///////////
// Structure for CtrlPcs Jema .  
//////////
TYPE PCS_Jema_IBX3 :
STRUCT
// PCS Controller  Measures
	AX_PowerCol					: ARRAY[1..3] OF PowerCol_Jema;

	MesData						: PCS ; 
	
	
	MesNbPowerCol_FreqReg			: UINT  ; (*(NA) Number of Power Column doing frequency regulation *)
	MesState_SoCLimitReached		: BOOL ; (*(NA) PCS SoC Limits has been reached *)
	MesHumidity						: REAL ; (*(%) Humidity*)
	
	MesReadCompleted				: BOOL ; 
	
	OUT_CmdBlackStart			: BOOL ; (* (NA) Blackstart Command *) 
	OUT_CmdGridMode				: BOOL ; (* (NA) Grid Mode Command *) 
	OUT_CmdP					: BOOL ; (* (NA) P setpoint regulation Mode Command *) 
	
	OUT_CmdQ				: BOOL ; (* (NA) Q setpoint regulation Mode Command *) 
	OUT_SetptV				: REAL ; (* (V) Voltage Reference for offgrid Mode *) 
	OUT_SetptCosPhi			: REAL ; (* (p.u) Cosphi Reference for Cosphi reg Mode *) 
	
	OUT_SetptF				: REAL ; 	(* (Hz) Frequency Reference for offgrid Mode *) 
	OUT_CmdCosPhi			: BOOL ; (* (NA) Cosphi regulation Mode Command *) 
	OUT_CmdUregMode			: BOOL ; (* (NA) Voltage Regulation Mode Command *) 
	OUT_CmdFreqregMode	: BOOL ; (* (NA) Frequency Regulation Mode Command *) 
END_STRUCT
END_TYPE

(* stored: Version 1.1.0.1, ProductVersion 3.1.4024.12
   DUT PCS_Jema_IBX3: Id {e14dc06c-e55c-4281-8cf1-e3bfd6fc2aff} *)
